// TIA Portal V16 export
// export: Created 2022-09-01T14:26:53.6763379Z, ExportSetting WithDefaults, DisplayName Totally Integrated Automation Portal, DisplayVersion V16, DisplayName TIA Portal Version Control Interface, DisplayVersion V16, DisplayName TIA Portal Openness, DisplayVersion V16, DisplayName STEP 7 Professional, DisplayVersion V16, DisplayName STEP 7 Safety, DisplayVersion V16, DisplayName WinCC Advanced, DisplayVersion V16
FUNCTION "Saídas_Bombas_Temporário" : Void   // FC17, LAD
{ S7_Optimized_Access := 'TRUE' }
VERSION : 0.1
// stored: AutoNumber true, IsIECCheckEnabled false, SetENOAutomatically false, UDAEnableTagReadback false
BEGIN

REGION Network 1
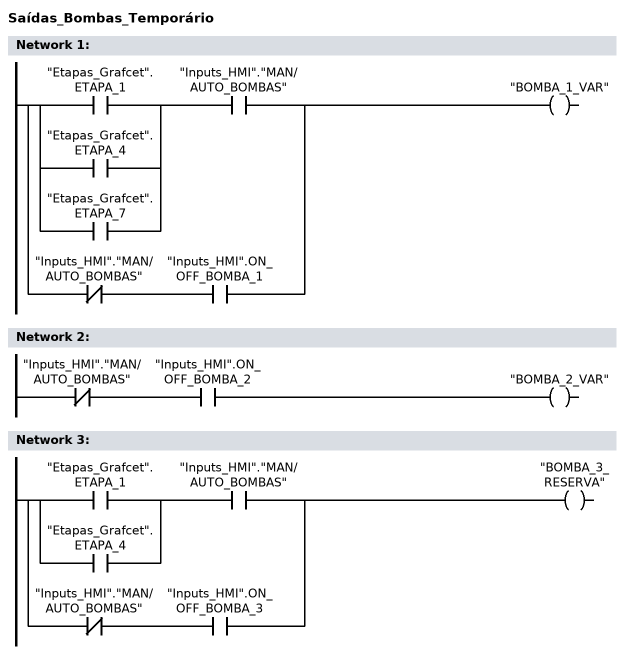
   RUNG wire#powerrail
      Contact( "Etapas_Grafcet".ETAPA_1 )
      wire#w1
      Contact( "Inputs_HMI"."MAN/AUTO_BOMBAS" )
      wire#w2
      Coil( "BOMBA_1_VAR" )
   END_RUNG
   RUNG wire#powerrail
      Contact( "Etapas_Grafcet".ETAPA_4 )
   END_RUNG wire#w1
   RUNG wire#powerrail
      Contact( "Etapas_Grafcet".ETAPA_7 )
   END_RUNG wire#w1
   RUNG wire#powerrail
      I_Contact( "Inputs_HMI"."MAN/AUTO_BOMBAS" )
      Contact( "Inputs_HMI".ON_OFF_BOMBA_1 )
   END_RUNG wire#w2
   // the same network as SCL:
   "BOMBA_1_VAR" := (("Etapas_Grafcet".ETAPA_1 OR "Etapas_Grafcet".ETAPA_4 OR "Etapas_Grafcet".ETAPA_7) AND "Inputs_HMI"."MAN/AUTO_BOMBAS") OR (NOT "Inputs_HMI"."MAN/AUTO_BOMBAS" AND "Inputs_HMI".ON_OFF_BOMBA_1);
END_REGION

REGION Network 2
   RUNG wire#powerrail
      I_Contact( "Inputs_HMI"."MAN/AUTO_BOMBAS" )
      Contact( "Inputs_HMI".ON_OFF_BOMBA_2 )
      Coil( "BOMBA_2_VAR" )
   END_RUNG
   // the same network as SCL:
   "BOMBA_2_VAR" := NOT "Inputs_HMI"."MAN/AUTO_BOMBAS" AND "Inputs_HMI".ON_OFF_BOMBA_2;
END_REGION

REGION Network 3
   RUNG wire#powerrail
      Contact( "Etapas_Grafcet".ETAPA_1 )
      wire#w1
      Contact( "Inputs_HMI"."MAN/AUTO_BOMBAS" )
      wire#w2
      Coil( "BOMBA_3_RESERVA" )
   END_RUNG
   RUNG wire#powerrail
      Contact( "Etapas_Grafcet".ETAPA_4 )
   END_RUNG wire#w1
   RUNG wire#powerrail
      I_Contact( "Inputs_HMI"."MAN/AUTO_BOMBAS" )
      Contact( "Inputs_HMI".ON_OFF_BOMBA_3 )
   END_RUNG wire#w2
   // the same network as SCL:
   "BOMBA_3_RESERVA" := (("Etapas_Grafcet".ETAPA_1 OR "Etapas_Grafcet".ETAPA_4) AND "Inputs_HMI"."MAN/AUTO_BOMBAS") OR (NOT "Inputs_HMI"."MAN/AUTO_BOMBAS" AND "Inputs_HMI".ON_OFF_BOMBA_3);
END_REGION
END_FUNCTION
